// TIA Portal V20 export
FUNCTION_BLOCK "FB_CmdCylinder"   // FB44, SCL
{ S7_Optimized_Access := 'TRUE' }
// stored: AutoNumber false, MemoryReserve 100, SetENOAutomatically false
   VAR_INPUT
      iEMinus { ExternalAccessible := 'False'; ExternalVisible := 'False'; ExternalWritable := 'False'} : Bool;
      iEPlus { ExternalAccessible := 'False'; ExternalVisible := 'False'; ExternalWritable := 'False'} : Bool;
      iMinusCmd { ExternalAccessible := 'False'; ExternalVisible := 'False'; ExternalWritable := 'False'} : Bool;
      iPlusCmd { ExternalAccessible := 'False'; ExternalVisible := 'False'; ExternalWritable := 'False'} : Bool;
      iJOGCmd { ExternalAccessible := 'False'; ExternalVisible := 'False'; ExternalWritable := 'False'} : Bool;
      iMonitorTime : Time;
   END_VAR
   VAR_OUTPUT
      oMinusPos { ExternalAccessible := 'False'; ExternalVisible := 'False'; ExternalWritable := 'False'} : Bool;
      oMiddlePos { ExternalAccessible := 'False'; ExternalVisible := 'False'; ExternalWritable := 'False'} : Bool;
      oPlusPos { ExternalAccessible := 'False'; ExternalVisible := 'False'; ExternalWritable := 'False'} : Bool;
      oErrorCode { ExternalAccessible := 'False'; ExternalVisible := 'False'; ExternalWritable := 'False'} : Int;
   END_VAR
   VAR_IN_OUT
      ioQMinus { ExternalAccessible := 'False'; ExternalVisible := 'False'; ExternalWritable := 'False'} : Bool;
      ioQPlus { ExternalAccessible := 'False'; ExternalVisible := 'False'; ExternalWritable := 'False'} : Bool;
   END_VAR
   VAR
      sRT_NoCmd : R_TRIG;
      sMonitorTimer { S7_SetPoint := 'True'} : TON_TIME;
   END_VAR
BEGIN
   REGION Description header 
       //==================================================================================
       // POSALUX Swiss SA / (C) Copyright 2025
       //----------------------------------------------------------------------------------
       // Title: FB_CmdCylinder
       // Comment/Function: Cylinder management with 2 outputs (Cmd) and two inputs (Pos)
       //                   Movements and positions are monitored:
       //                      Error Code 0: No Error
       //                      Error Code 1: Error Timeout Command Plus
       //                      Error Code 2: Error Timeout Command Minus
       //                      Error Code 3: Error Timeout Position OFF   
       //                      Error Code 4: Error Timeout Position ON             
       // Author: Fabien WALDT
       // Engineering: TIA Portal v17
       //----------------------------------------------------------------------------------
       // Change log table:
       // Version  | Date     | Expert in charge | Changes applied
       // ---------|----------|------------------|-----------------------------------------
       // 00.00.01 | 20250501 | WFA              | First released version
       // =================================================================================
   END_REGION

   REGION Init
       // No command : both plus and minus are set. (WFA ??)
       #sRT_NoCmd(CLK:=NOT #ioQMinus AND NOT #ioQPlus);
       IF #sRT_NoCmd.Q THEN
           #ioQMinus := TRUE;
           #ioQPlus := TRUE;
           RETURN;
       END_IF;
   END_REGION

   REGION Plus / Minus Commands
       // Minus Command
       IF #iMinusCmd THEN
           #ioQPlus := FALSE;
           #ioQMinus := TRUE;
       END_IF;

       // Plus Command
       IF #iPlusCmd THEN
           #ioQMinus := FALSE;
           #ioQPlus := TRUE;
       END_IF;

       // JOG stop on the way : both plus and minus are set. (WFA ??)
       IF #iJOGCmd AND NOT #iMinusCmd AND NOT #iPlusCmd THEN
           #ioQMinus := TRUE;
           #ioQPlus := TRUE;
       END_IF;
   END_REGION

   REGION Positions
       #oMinusPos := #iEMinus AND NOT #iEPlus;
       #oMiddlePos := NOT #iEMinus AND NOT #iEPlus;
       #oPlusPos := #iEPlus AND NOT #iEMinus;
   END_REGION

   REGION Monitoring Timer
       #sMonitorTimer(IN:=(#iMinusCmd AND NOT #oMinusPos) OR
                      (#iPlusCmd AND NOT #oPlusPos) OR
                      (NOT #oMinusPos AND NOT #oPlusPos) OR
                      (#iEMinus AND #iEPlus),
                      PT:=#iMonitorTime);
   END_REGION

   REGION Error Codes
       #oErrorCode := 0;           // Code 0: No Error
       IF #iPlusCmd AND #sMonitorTimer.Q THEN
           #oErrorCode := 1;       // Code 1: Error Timeout Command Plus
       ELSIF #iMinusCmd AND #sMonitorTimer.Q THEN
           #oErrorCode := 2;       // Code 2: Error Timeout Command Minus
       ELSIF NOT #oMinusPos AND NOT #oPlusPos AND #sMonitorTimer.Q THEN
           #oErrorCode := 3;       // Code 3: Error Timeout Position OFF   
       ELSIF #iEMinus AND #iEPlus AND #sMonitorTimer.Q THEN
           #oErrorCode := 4;       // Code 4: Error Timeout Position ON       
       END_IF;
   END_REGION
END_FUNCTION_BLOCK
